% RSLogix 500 project CAM_OPERATED_CONTROL_VALVE.RSS, saved by version 8.30.00.16 %
PROJECT "PROC1"    % processor: Bul.1763 MicroLogix 1100 Series B %

PROGRAM FILES
  LAD 2   5 rungs
  LAD 3 "IO"  7 rungs
  LAD 4 "POSITION"  6 rungs
  LAD 5 "CYCLES"  10 rungs
  LAD 6 "CONTROLS"  2 rungs

DATA FILES
  O0 OUTPUT  4 elements
  I1 INPUT  6 elements
  S2 STATUS  66 elements
  B3 BINARY  5 elements
  T4 TIMER  3 elements
  C5 COUNTER  1 elements
  R6 CONTROL  1 elements
  N7 INTEGER  2 elements
  F8 FLOAT  1 elements

LADDER 2
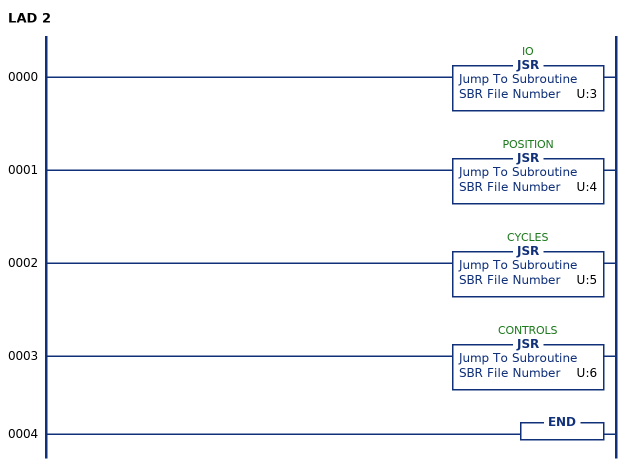
% Rung: 0 %
SOR JSR U:3 EOR
%   U:3  "IO" %
% Rung: 1 %
SOR JSR U:4 EOR
%   U:4  "POSITION" %
% Rung: 2 %
SOR JSR U:5 EOR
%   U:5  "CYCLES" %
% Rung: 3 %
SOR JSR U:6 EOR
%   U:6  "CONTROLS" %
% Rung: 4 %
SOR END EOR

LADDER 3 "IO"
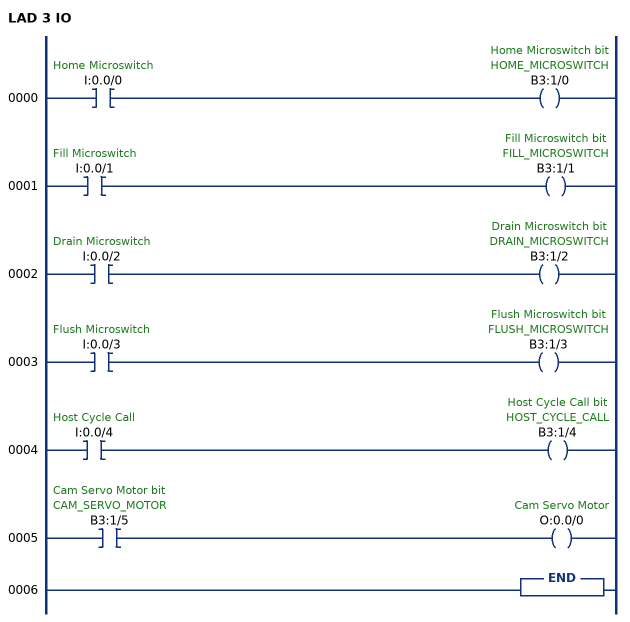
% Rung: 0 %
SOR XIC I:0.0/0 OTE B3:1/0 EOR
%   I:0.0/0  "Home Microswitch" %
%   B3:1/0  HOME_MICROSWITCH  "Home Microswitch bit" %
% Rung: 1 %
SOR XIC I:0.0/1 OTE B3:1/1 EOR
%   I:0.0/1  "Fill Microswitch" %
%   B3:1/1  FILL_MICROSWITCH  "Fill Microswitch bit" %
% Rung: 2 %
SOR XIC I:0.0/2 OTE B3:1/2 EOR
%   I:0.0/2  "Drain Microswitch" %
%   B3:1/2  DRAIN_MICROSWITCH  "Drain Microswitch bit" %
% Rung: 3 %
SOR XIC I:0.0/3 OTE B3:1/3 EOR
%   I:0.0/3  "Flush Microswitch" %
%   B3:1/3  FLUSH_MICROSWITCH  "Flush Microswitch bit" %
% Rung: 4 %
SOR XIC I:0.0/4 OTE B3:1/4 EOR
%   I:0.0/4  "Host Cycle Call" %
%   B3:1/4  HOST_CYCLE_CALL  "Host Cycle Call bit" %
% Rung: 5 %
SOR XIC B3:1/5 OTE O:0.0/0 EOR
%   B3:1/5  CAM_SERVO_MOTOR  "Cam Servo Motor bit" %
%   O:0.0/0  "Cam Servo Motor" %
% Rung: 6 %
SOR END EOR

LADDER 4 "POSITION"
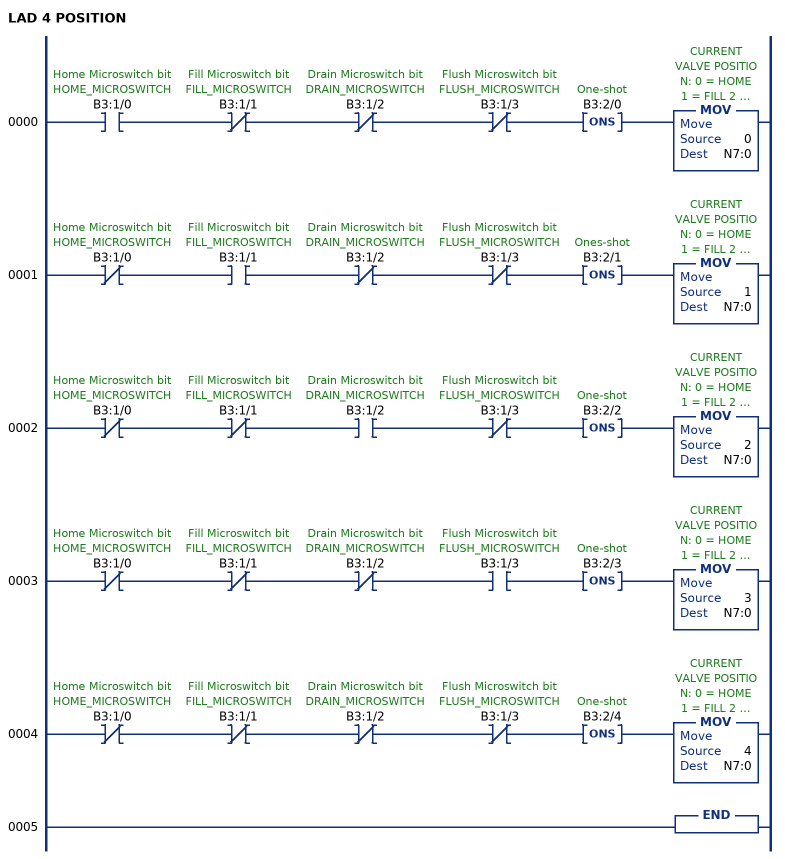
% Rung: 0 %
SOR XIC B3:1/0 XIO B3:1/1 XIO B3:1/2 XIO B3:1/3 ONS B3:2/0 MOV 0 N7:0 EOR
%   B3:1/0  HOME_MICROSWITCH  "Home Microswitch bit" %
%   B3:1/1  FILL_MICROSWITCH  "Fill Microswitch bit" %
%   B3:1/2  DRAIN_MICROSWITCH  "Drain Microswitch bit" %
%   B3:1/3  FLUSH_MICROSWITCH  "Flush Microswitch bit" %
%   B3:2/0  "One-shot" %
%   N7:0  "CURRENT VALVE POSITION: 0 = HOME   1 = FILL 2 = DRAIN  3 = FLUSH 4 = TRAVEL" %
% Rung: 1 %
SOR XIO B3:1/0 XIC B3:1/1 XIO B3:1/2 XIO B3:1/3 ONS B3:2/1 MOV 1 N7:0 EOR
%   B3:1/0  HOME_MICROSWITCH  "Home Microswitch bit" %
%   B3:1/1  FILL_MICROSWITCH  "Fill Microswitch bit" %
%   B3:1/2  DRAIN_MICROSWITCH  "Drain Microswitch bit" %
%   B3:1/3  FLUSH_MICROSWITCH  "Flush Microswitch bit" %
%   B3:2/1  "Ones-shot" %
%   N7:0  "CURRENT VALVE POSITION: 0 = HOME   1 = FILL 2 = DRAIN  3 = FLUSH 4 = TRAVEL" %
% Rung: 2 %
SOR XIO B3:1/0 XIO B3:1/1 XIC B3:1/2 XIO B3:1/3 ONS B3:2/2 MOV 2 N7:0 EOR
%   B3:1/0  HOME_MICROSWITCH  "Home Microswitch bit" %
%   B3:1/1  FILL_MICROSWITCH  "Fill Microswitch bit" %
%   B3:1/2  DRAIN_MICROSWITCH  "Drain Microswitch bit" %
%   B3:1/3  FLUSH_MICROSWITCH  "Flush Microswitch bit" %
%   B3:2/2  "One-shot" %
%   N7:0  "CURRENT VALVE POSITION: 0 = HOME   1 = FILL 2 = DRAIN  3 = FLUSH 4 = TRAVEL" %
% Rung: 3 %
SOR XIO B3:1/0 XIO B3:1/1 XIO B3:1/2 XIC B3:1/3 ONS B3:2/3 MOV 3 N7:0 EOR
%   B3:1/0  HOME_MICROSWITCH  "Home Microswitch bit" %
%   B3:1/1  FILL_MICROSWITCH  "Fill Microswitch bit" %
%   B3:1/2  DRAIN_MICROSWITCH  "Drain Microswitch bit" %
%   B3:1/3  FLUSH_MICROSWITCH  "Flush Microswitch bit" %
%   B3:2/3  "One-shot" %
%   N7:0  "CURRENT VALVE POSITION: 0 = HOME   1 = FILL 2 = DRAIN  3 = FLUSH 4 = TRAVEL" %
% Rung: 4 %
SOR XIO B3:1/0 XIO B3:1/1 XIO B3:1/2 XIO B3:1/3 ONS B3:2/4 MOV 4 N7:0 EOR
%   B3:1/0  HOME_MICROSWITCH  "Home Microswitch bit" %
%   B3:1/1  FILL_MICROSWITCH  "Fill Microswitch bit" %
%   B3:1/2  DRAIN_MICROSWITCH  "Drain Microswitch bit" %
%   B3:1/3  FLUSH_MICROSWITCH  "Flush Microswitch bit" %
%   B3:2/4  "One-shot" %
%   N7:0  "CURRENT VALVE POSITION: 0 = HOME   1 = FILL 2 = DRAIN  3 = FLUSH 4 = TRAVEL" %
% Rung: 5 %
SOR END EOR

LADDER 5 "CYCLES"
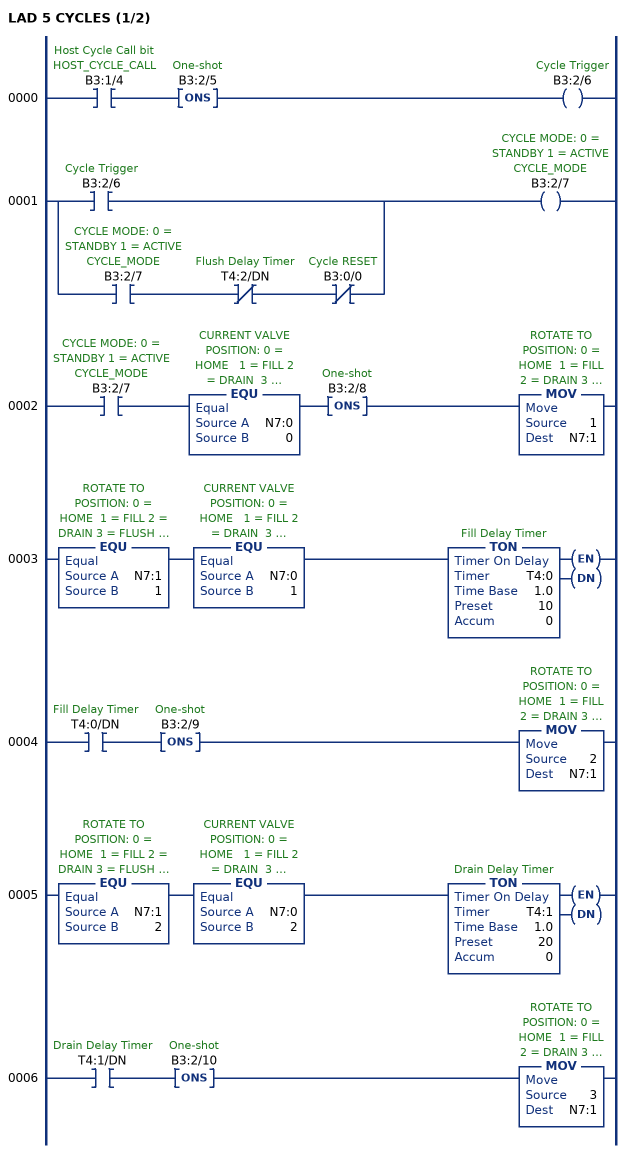
% Rung: 0 %
SOR XIC B3:1/4 ONS B3:2/5 OTE B3:2/6 EOR
%   B3:1/4  HOST_CYCLE_CALL  "Host Cycle Call bit" %
%   B3:2/5  "One-shot" %
%   B3:2/6  "Cycle Trigger" %
% Rung: 1 %
SOR BST XIC B3:2/6 NXB XIC B3:2/7 XIO T4:2/DN XIO B3:0/0 BND OTE B3:2/7 EOR
%   B3:2/6  "Cycle Trigger" %
%   B3:2/7  CYCLE_MODE  "CYCLE MODE: 0 = STANDBY 1 = ACTIVE" %
%   T4:2  "Flush Delay Timer" %
%   B3:0/0  "Cycle RESET" %
% Rung: 2 %
SOR XIC B3:2/7 EQU N7:0 0 ONS B3:2/8 MOV 1 N7:1 EOR
%   B3:2/7  CYCLE_MODE  "CYCLE MODE: 0 = STANDBY 1 = ACTIVE" %
%   N7:0  "CURRENT VALVE POSITION: 0 = HOME   1 = FILL 2 = DRAIN  3 = FLUSH 4 = TRAVEL" %
%   B3:2/8  "One-shot" %
%   N7:1  "ROTATE TO POSITION: 0 = HOME  1 = FILL 2 = DRAIN 3 = FLUSH 4 = TRAVEL" %
% Rung: 3 %
SOR EQU N7:1 1 EQU N7:0 1 TON T4:0 1.0 10 0 EOR
%   N7:1  "ROTATE TO POSITION: 0 = HOME  1 = FILL 2 = DRAIN 3 = FLUSH 4 = TRAVEL" %
%   N7:0  "CURRENT VALVE POSITION: 0 = HOME   1 = FILL 2 = DRAIN  3 = FLUSH 4 = TRAVEL" %
%   T4:0  "Fill Delay Timer" %
% Rung: 4 %
SOR XIC T4:0/DN ONS B3:2/9 MOV 2 N7:1 EOR
%   T4:0  "Fill Delay Timer" %
%   B3:2/9  "One-shot" %
%   N7:1  "ROTATE TO POSITION: 0 = HOME  1 = FILL 2 = DRAIN 3 = FLUSH 4 = TRAVEL" %
% Rung: 5 %
SOR EQU N7:1 2 EQU N7:0 2 TON T4:1 1.0 20 0 EOR
%   N7:1  "ROTATE TO POSITION: 0 = HOME  1 = FILL 2 = DRAIN 3 = FLUSH 4 = TRAVEL" %
%   N7:0  "CURRENT VALVE POSITION: 0 = HOME   1 = FILL 2 = DRAIN  3 = FLUSH 4 = TRAVEL" %
%   T4:1  "Drain Delay Timer" %
% Rung: 6 %
SOR XIC T4:1/DN ONS B3:2/10 MOV 3 N7:1 EOR
%   T4:1  "Drain Delay Timer" %
%   B3:2/10  "One-shot" %
%   N7:1  "ROTATE TO POSITION: 0 = HOME  1 = FILL 2 = DRAIN 3 = FLUSH 4 = TRAVEL" %

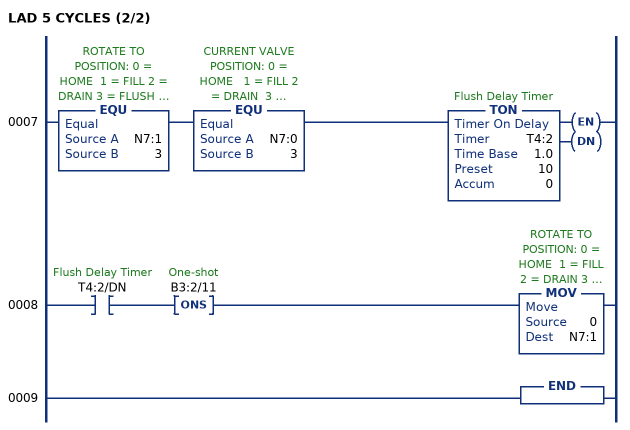
% Rung: 7 %
SOR EQU N7:1 3 EQU N7:0 3 TON T4:2 1.0 10 0 EOR
%   N7:1  "ROTATE TO POSITION: 0 = HOME  1 = FILL 2 = DRAIN 3 = FLUSH 4 = TRAVEL" %
%   N7:0  "CURRENT VALVE POSITION: 0 = HOME   1 = FILL 2 = DRAIN  3 = FLUSH 4 = TRAVEL" %
%   T4:2  "Flush Delay Timer" %
% Rung: 8 %
SOR XIC T4:2/DN ONS B3:2/11 MOV 0 N7:1 EOR
%   T4:2  "Flush Delay Timer" %
%   B3:2/11  "One-shot" %
%   N7:1  "ROTATE TO POSITION: 0 = HOME  1 = FILL 2 = DRAIN 3 = FLUSH 4 = TRAVEL" %
% Rung: 9 %
SOR END EOR

LADDER 6 "CONTROLS"
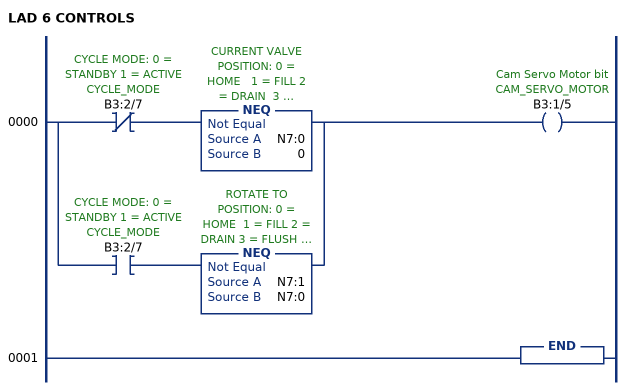
% Rung: 0 %
SOR BST XIO B3:2/7 NEQ N7:0 0 NXB XIC B3:2/7 NEQ N7:1 N7:0 BND OTE B3:1/5 EOR
%   B3:2/7  CYCLE_MODE  "CYCLE MODE: 0 = STANDBY 1 = ACTIVE" %
%   N7:0  "CURRENT VALVE POSITION: 0 = HOME   1 = FILL 2 = DRAIN  3 = FLUSH 4 = TRAVEL" %
%   N7:1  "ROTATE TO POSITION: 0 = HOME  1 = FILL 2 = DRAIN 3 = FLUSH 4 = TRAVEL" %
%   B3:1/5  CAM_SERVO_MOTOR  "Cam Servo Motor bit" %
% Rung: 1 %
SOR END EOR

DATA TABLE (non-zero values as saved)
DATA B3
% B3:0 % 0X0000 0X0020 0X0010 0X0000 0X0000
DATA T4
% .PRE .ACC %
% T4:0 % 10 0
% T4:1 % 20 0
% T4:2 % 10 0
DATA N7
% N7:0 % 4 1
